FUNCTION_BLOCK MissingKeyDeserializationError_TestSuite EXTENDS TcUnit.FB_TestSuite

TestAccept();
TestErrorType();
TestIsSameAsWithSameErrors();
TestIsSameAsWithDifferentErrors();
TestMessage();
TestSerializeWith();

METHOD PUBLIC TestAccept
VAR
	error : MissingKeyDeserializationError('testKey');
	visitor : MockVisitor(ExpectedError := error);
END_VAR
TEST('TestAccept');

error.Accept(visitor);

AssertTrue(
	Condition := visitor.VisitedCorrectError,
	Message := 'Did not invoke VisitError on the visitor'
);

TEST_FINISHED();
END_METHOD

METHOD PUBLIC TestErrorType
VAR
	error : MissingKeyDeserializationError('testKey');
END_VAR
TEST('TestErrorType');

AssertEquals_String(
	Actual := error.ErrorType,
	Expected := 'MISSING_KEY_DESERIALIZATION_ERROR',
	Message := 'Did not return the expected ErrorType'
);

TEST_FINISHED();
END_METHOD

METHOD PUBLIC TestIsSameAsWithDifferentErrors
VAR
	error1 : MissingKeyDeserializationError('testKey');
	error2 : MockError(MockErrorType:='ERROR_TYPE_B',MockMessage:='Message 2');
END_VAR
TEST('TestIsSameAsWithDifferentErrors');

AssertFalse(
	Condition := error1.IsSameAs(error2),
	Message := 'Did not correctly identify errors as being different type'
);

TEST_FINISHED();
END_METHOD

METHOD PUBLIC TestIsSameAsWithSameErrors
VAR
	error1 : MissingKeyDeserializationError('testKey');
	error2 : MockError(MockErrorType:='MISSING_KEY_DESERIALIZATION_ERROR',MockMessage:='Message');
END_VAR
TEST('TestIsSameAsWithSameErrors');

AssertTrue(
	Condition := error1.IsSameAs(error2),
	Message := 'Did not correctly identify errors as being the same type'
);

TEST_FINISHED();
END_METHOD

METHOD PUBLIC TestMessage
VAR
	error : MissingKeyDeserializationError('testKey');
END_VAR
TEST('TestMessage');

AssertEquals_String(
	Actual := error.Message,
	Expected := 'Deserialization Failed, Missing Key : testKey',
	Message := 'Did not return the expected Message'
);

TEST_FINISHED();
END_METHOD

METHOD PUBLIC TestSerializeWith
VAR
	error : MissingKeyDeserializationError('testKey');
	serializer : JsonSerializer;
	result : T_MAXSTRING;
END_VAR
TEST('TestSerializeWith');

error.SerializeWith(serializer);
serializer.TryGetSerializedData(ADR(result), SIZEOF(result));

AssertEquals_String(
	Actual := result,
	Expected := '{"errorType":"MISSING_KEY_DESERIALIZATION_ERROR","message":"Deserialization Failed, Missing Key : testKey"}',
	Message := 'Did not serialize correctly'
);

TEST_FINISHED();
END_METHOD

END_FUNCTION_BLOCK

(* stored: Version 1.1.0.1, ProductVersion 3.1.4024.12
   POU MissingKeyDeserializationError_TestSuite: Id {b70e347a-a69b-081e-1f13-52157cf195c9}, SpecialFunc None
   Method TestAccept: Id {a76fda00-c17c-077d-0913-cd48d512f9d2}
   Method TestErrorType: Id {c3e791f1-eff7-0d7b-3182-1a70d2f3ef41}
   Method TestIsSameAsWithDifferentErrors: Id {dd37ab02-163c-07f5-3940-73b2098ae3d9}
   Method TestIsSameAsWithSameErrors: Id {ef536c4e-ebb4-0814-255c-8383c5789de8}
   Method TestMessage: Id {9e00e1c0-1e29-08c9-0d4f-5c8d250fd37c}
   Method TestSerializeWith: Id {841393e8-db5d-0bc9-3555-594488606e4c} *)
